{attribute 'GeneratedUsingTerminal: EL7041-0001-0016'}
{attribute addProperty BoxType "EL7041-0001-0016"}
{attribute addProperty Id "StatusAT %I*Status_36C8BFF110"}
{attribute addProperty CRC "1532699765"}
{attribute addProperty Size "10"}
TYPE STM_Status_5B5B2475 EXTENDS InputBase_8311D824 :
STRUCT
	{attribute addProperty Name "Status"}
	Status AT %I* : Status_36C8BFF1;
END_STRUCT
END_TYPE

(* stored: Version 1.2.0.0, ProductVersion 3.1.4024.9
   DUT STM_Status_5B5B2475: Id {8ec0350c-26b5-4606-b89b-5562d5c5d05c} *)
